FUNCTION_BLOCK MoveVelocity IMPLEMENTS I_Task
VAR
	mcMoveVelo : MC_MoveVelocity;
	_Axis : REFERENCE TO Tc2_MC2.AXIS_REF;
	_MoveAtVelo : BOOL;
	State: INT;
	_Done: BOOL;
	_Error: BOOL;
	_Busy: BOOL;
END_VAR

METHOD Abort : BOOL
mcMoveVelo.Execute := FALSE;
_Busy := FALSE;
_MoveAtVelo := FALSE;
Abort := TRUE;
State := 0;
END_METHOD

PROPERTY PUBLIC Acceleration : mc_lreal
GET
Acceleration := mcMoveVelo.Acceleration;
END_GET
SET
mcMoveVelo.Acceleration := Acceleration;
mcMoveVelo.Acceleration := Acceleration;
END_SET
END_PROPERTY

PROPERTY Busy : BOOL
GET
Busy := _Busy;
END_GET
END_PROPERTY

METHOD Cycle : HRESULT
Cycle := S_OK;
CASE State OF
	0:
		IF _MoveAtVelo THEN
			Cycle := S_PENDING;
			_Done := FALSE;
			_Error := FALSE;
			_Busy := TRUE;
			mcMoveVelo.Execute := TRUE;
			IF mcMoveVelo.Busy THEN
				State := 10;
				_MoveAtVelo := FALSE;
			END_IF
		END_IF
	
	10:
		IF NOT mcMoveVelo.Busy THEN
			IF mcMoveVelo.InVelocity THEN
				_Done := TRUE;
			ELSIF mcMoveVelo.Error THEN
				_Error := TRUE;
			END_IF
			_Busy := FALSE;
			mcMoveVelo.Execute := FALSE;
			State := 0;
			Cycle := S_OK;
		END_IF
	ELSE
		Cycle := E_FAIL;
END_CASE

mcMoveVelo(Axis := _Axis);
END_METHOD

PROPERTY Deceleration : MC_LREAL
GET
Deceleration := mcMoveVelo.Deceleration;
END_GET
SET
mcMoveVelo.Deceleration := Deceleration;
END_SET
END_PROPERTY

PROPERTY Done : BOOL
GET
Done := _Done;
END_GET
END_PROPERTY

PROPERTY Error : BOOL
GET
Error := _Error;
END_GET
END_PROPERTY

//FB_Init is always available implicitly and it is used primarily for initialization.
//The return value is not evaluated. For a specific influence, you can also declare the
//methods explicitly and provide additional code there with the standard initialization
//code. You can evaluate the return value.
METHOD FB_Init: BOOL
VAR_INPUT
    bInitRetains: BOOL; // TRUE: the retain variables are initialized (reset warm / reset cold)
    bInCopyCode: BOOL;  // TRUE: the instance will be copied to the copy code afterward (online change)   
	axis : reference TO AXIS_REF;
END_VAR
_Axis REF= axis;
END_METHOD

PROPERTY Jerk : MC_LREAL
GET
Jerk := mcMoveVelo.Jerk;
END_GET
SET
mcMoveVelo.Jerk := Jerk;
END_SET
END_PROPERTY

METHOD MoveAtVelocity : HRESULT
VAR_INPUT
	Direction : MC_Direction;
	Velocity : MC_LREAL;
	Task : REFERENCE TO I_Task;
END_VAR
IF Velocity = 0 THEN
	MoveAtVelocity := -1;
	RETURN;
END_IF

mcMoveVelo.Direction := Direction;
mcMoveVelo.Velocity := Velocity;
MoveAtVelocity := 1;
_MoveAtVelo := TRUE;
Task := THIS^;
END_METHOD

END_FUNCTION_BLOCK

(* stored: Version 1.1.0.1
   POU MoveVelocity: Id {86fa777b-f5d3-4d7e-bd44-8ee6f4991e5f}, SpecialFunc None
   Method Abort: Id {24ef1d79-00e6-485e-b5bc-96b2e835c968}
   Property Acceleration: Id {5690795c-3a83-420b-9da3-878026ded205}
   Get Get: Id {40d0149e-7955-4b29-bb76-c9562232dbff}
   Set Set: Id {7266777e-dab1-408a-acab-1fd1c86a3fb1}
   Property Busy: Id {412e554f-b115-468a-8039-f1c3519a13a0}
   Get Get: Id {0cd54035-de2e-4540-a890-85dbe5996ff8}
   Method Cycle: Id {3a4012ad-a672-409a-903c-5dab8269f3b3}
   Property Deceleration: Id {3687a92b-814f-4a65-b007-ae191bb9e61e}
   Get Get: Id {fd15208c-b78a-429b-9b89-acf251926f83}
   Set Set: Id {086f87de-d583-4d56-b50a-8d0c08599476}
   Property Done: Id {51dcd633-8b8c-4ebb-bd82-704ceec64f29}
   Get Get: Id {da58fae3-77f4-4bde-881d-5f11edd1c4f2}
   Property Error: Id {020f061a-cd8f-4d42-86c0-592c671fd6ba}
   Get Get: Id {396b9440-fb51-44e4-9398-6c6a1bb2ceb4}
   Method FB_Init: Id {a43ce224-e4a7-43b4-bb34-a8a929700026}
   Property Jerk: Id {47d3b6ef-be1c-4ef3-b364-6e63da359318}
   Get Get: Id {b6612f32-b3b3-4b77-9630-833953175823}
   Set Set: Id {4e83b889-5283-4cde-9447-b4b10940b51e}
   Method MoveAtVelocity: Id {1db16ae1-c549-47f3-8cc7-5298e04ee848} *)
